% RSLogix 500 project Saw Mill.RSS, saved by version 8.30.00.16 %
PROJECT "UNTITLED"    % processor: Bul.1763 MicroLogix 1100 Series B %

PROGRAM FILES
  LAD 2   6 rungs

DATA FILES
  O0 OUTPUT  4 elements
  I1 INPUT  6 elements
  S2 STATUS  66 elements
  B3 BINARY  1 elements
  T4 TIMER  20 elements
  C5 COUNTER  1 elements
  R6 CONTROL  1 elements
  N7 INTEGER  1 elements
  F8 FLOAT  1 elements

LADDER 2
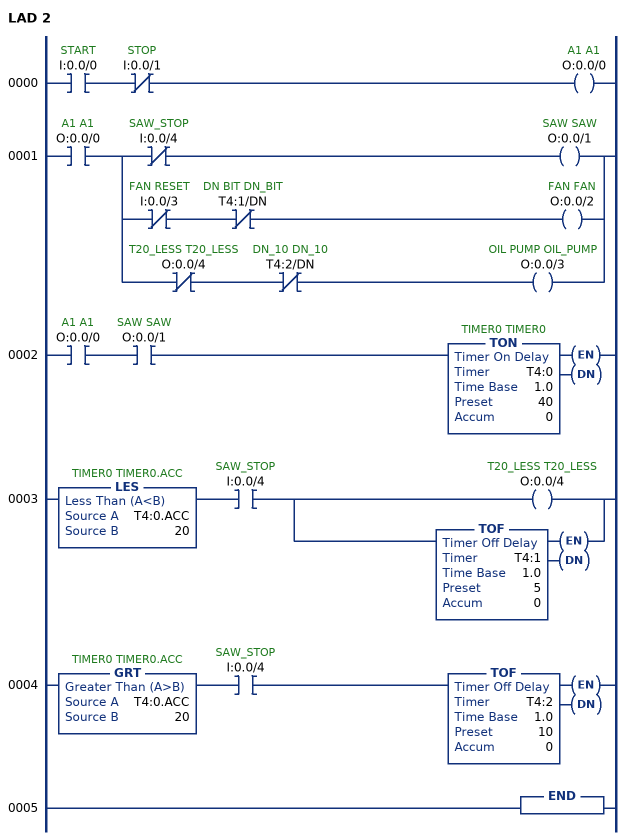
% Rung: 0 %
SOR XIC I:0.0/0 XIO I:0.0/1 OTE O:0.0/0 EOR
%   I:0.0/0  "START" %
%   I:0.0/1  "STOP" %
%   O:0.0/0  A1  "A1" %
% Rung: 1 %
SOR XIC O:0.0/0 BST BST XIO I:0.0/4 OTE O:0.0/1 NXB XIO I:0.0/3 XIO T4:1/DN OTE O:0.0/2 BND NXB XIO O:0.0/4 XIO T4:2/DN OTE O:0.0/3 BND EOR
%   O:0.0/0  A1  "A1" %
%   I:0.0/4  "SAW_STOP" %
%   O:0.0/1  SAW  "SAW" %
%   I:0.0/3  "FAN RESET" %
%   T4:1/DN  DN_BIT  "DN BIT" %
%   O:0.0/2  FAN  "FAN" %
%   O:0.0/4  T20_LESS  "T20_LESS" %
%   T4:2/DN  DN_10  "DN_10" %
%   O:0.0/3  OIL_PUMP  "OIL PUMP" %
% Rung: 2 %
SOR XIC O:0.0/0 XIC O:0.0/1 TON T4:0 1.0 40 0 EOR
%   O:0.0/0  A1  "A1" %
%   O:0.0/1  SAW  "SAW" %
%   T4:0  TIMER0  "TIMER0" %
% Rung: 3 %
SOR LES T4:0.ACC 20 XIC I:0.0/4 BST OTE O:0.0/4 NXB TOF T4:1 1.0 5 0 BND EOR
%   T4:0  TIMER0  "TIMER0" %
%   I:0.0/4  "SAW_STOP" %
%   O:0.0/4  T20_LESS  "T20_LESS" %
% Rung: 4 %
SOR GRT T4:0.ACC 20 XIC I:0.0/4 TOF T4:2 1.0 10 0 EOR
%   T4:0  TIMER0  "TIMER0" %
%   I:0.0/4  "SAW_STOP" %
% Rung: 5 %
SOR END EOR

OTHER DOCUMENTED ADDRESSES
  I:0  INPUT  "input"
  I:0.0/2  "A1"
  I:0.1/0  STOP  "STOP"
  I:1  START1  "start"
  I:1.0  START  "Start"
  I:1.0/0  "INPUT"
  N7:0  TWENTY  "twenty seconds"
  O:0  OUTPUT  "OUTPUT"
  O:0.0/5  T20_MORE  "T20 MORE"
  O:1  OUTPUT1  "OUTPUT"
  O:1.0  OUTPU1  "Output"
  O:1.0/0  "OUTPUT"

DATA TABLE (non-zero values as saved)
DATA T4
% .PRE .ACC %
% T4:0 % 40 0
% T4:1 % 5 0
% T4:2 % 10 0
DATA N7
% N7:0 % 20
